{attribute 'GeneratedUsingTerminal: AMP8000-0030-0103-0103'}
{attribute addProperty BoxType "AMP8000-0030-0103-0103"}
{attribute addProperty Id "FSoE_Master_CmdUSINT1Axis_A_STOBOOL1Safe_Output_1BOOL1Safe_Output_2BOOL1Safe_Output_3BOOL1Safe_Output_4BOOL1Safe_Output_5BOOL1Safe_Output_6BOOL1Safe_Output_7BOOL1Axis_B_STOBOOL1Safe_Output_9BOOL1Safe_Output_10BOOL1Safe_Output_11BOOL1Safe_Output_12BOOL1Safe_Output_13BOOL1Safe_Output_14BOOL1Safe_Output_15BOOL1FSoE_Master_CRC_0UINT2FSoE_Master_ConnIDUINT2"}
{attribute addProperty CRC "1786964883"}
{attribute addProperty Size "21"}
TYPE FSOE_6A82EB93 :
STRUCT
	{attribute addProperty Name "FSoE_Master_Cmd"}
	FSoE_Master_Cmd : USINT;
	{attribute addProperty Name "Axis_A_STO"}
	Axis_A_STO : BOOL;
	{attribute addProperty Name "Safe_Output_1"}
	Safe_Output_1 : BOOL;
	{attribute addProperty Name "Safe_Output_2"}
	Safe_Output_2 : BOOL;
	{attribute addProperty Name "Safe_Output_3"}
	Safe_Output_3 : BOOL;
	{attribute addProperty Name "Safe_Output_4"}
	Safe_Output_4 : BOOL;
	{attribute addProperty Name "Safe_Output_5"}
	Safe_Output_5 : BOOL;
	{attribute addProperty Name "Safe_Output_6"}
	Safe_Output_6 : BOOL;
	{attribute addProperty Name "Safe_Output_7"}
	Safe_Output_7 : BOOL;
	{attribute addProperty Name "Axis_B_STO"}
	Axis_B_STO : BOOL;
	{attribute addProperty Name "Safe_Output_9"}
	Safe_Output_9 : BOOL;
	{attribute addProperty Name "Safe_Output_10"}
	Safe_Output_10 : BOOL;
	{attribute addProperty Name "Safe_Output_11"}
	Safe_Output_11 : BOOL;
	{attribute addProperty Name "Safe_Output_12"}
	Safe_Output_12 : BOOL;
	{attribute addProperty Name "Safe_Output_13"}
	Safe_Output_13 : BOOL;
	{attribute addProperty Name "Safe_Output_14"}
	Safe_Output_14 : BOOL;
	{attribute addProperty Name "Safe_Output_15"}
	Safe_Output_15 : BOOL;
	{attribute addProperty Name "FSoE_Master_CRC_0"}
	FSoE_Master_CRC_0 : UINT;
	{attribute addProperty Name "FSoE_Master_ConnID"}
	FSoE_Master_ConnID : UINT;
END_STRUCT
END_TYPE

(* stored: Version 1.2.0.0, ProductVersion 3.1.4024.9
   DUT FSOE_6A82EB93: Id {93f9939d-73db-404c-bd2c-5366bf7ecad8} *)
